// TIA Portal V16 export
// export: Created 2022-11-17T15:49:49.7301291Z, ExportSetting WithDefaults, DisplayName Totally Integrated Automation Portal, DisplayVersion V16 Update 6, DisplayName TIA Portal Version Control Interface, DisplayVersion V16 Update 2, DisplayName TIA Portal Openness, DisplayVersion V16 Update 6, DisplayName SINAMICS Startdrive Advanced, DisplayVersion V16 Update 5, DisplayName SINAMICS Startdrive G130, G150, S120, S150, SINAMICS MV, S210, DisplayVersion V16 Update 5, DisplayName SINAMICS Startdrive G110M, G120, G120C, G120D, G120P, G115D, DisplayVersion V16 Update 5, DisplayName STEP 7 Professional, DisplayVersion V16 Update 6, DisplayName STEP 7 Safety, DisplayVersion V16, DisplayName WinCC Advanced, DisplayVersion V16 Update 6
TYPE "ProgramDataGreyBar"
// stored: IsFailsafeCompliant false
   STRUCT
      Overlap : Int;   // Film overlap
      Height : Int;   // Spool carriage height (mm)
      Landmark : Bool;   // Landmark (0=Bottom 1=Top)
      Lifter : Bool;   // Pallet lifter
      SpareBit1 : Bool;   // Spare
      Airblower : Bool;   // Airblower on film tail (0=Excluded 1=Included)
      NextStep : Bool;   // Next step (0=End 1=Next)
      PressureP : Bool;   // Pressure plate (0=Excluded 1=Included)
      SpareByte1 : Byte;   // Spare
      Revolution : Int;   // Revolutions
      RopeUnitUpper : Byte;   // Upper rope unit (1=Exc 2=Inc 3=Inc during)
      RopeUnitLower : Byte;   // Lower rope unit (1=Exc 2=Inc 3=Inc during)
      FilmForce : Int;   // Film force
      FilmPrestretch : Int;   // Film prestretch
      SpareWord1 : Int;   // Spare
      SpareWord2 : Int;   // Spare
      SpareWord3 : Int;   // Spare
      SpareWord4 : Int;   // Spare
      SpareWord5 : Int;   // Spare
      SpareWord6 : Int;   // Spare
   END_STRUCT;
END_TYPE
